// TIA Portal V17 export
// export: Created 2025-08-05T09:36:00.4025579Z, ExportSetting WithDefaults, DisplayName Totally Integrated Automation Portal, DisplayVersion V17, DisplayName TIA Portal Openness, DisplayVersion V17, DisplayName TIA Portal Version Control Interface, DisplayVersion V17, DisplayName SINAMICS Startdrive Advanced, DisplayVersion V17, DisplayName SINAMICS Startdrive G130, G150, S120, S150, SINAMICS MV, S210, DisplayVersion V17, DisplayName SINAMICS Startdrive G110M, G120, G120C, G120D, G120P, G115D, DisplayVersion V17, DisplayName STEP 7 Professional, DisplayVersion V17, DisplayName STEP 7 Safety, DisplayVersion V17, DisplayName WinCC Advanced, DisplayVersion V17
TYPE "typeHmiCounter"
TITLE = HMI part counter / HMI Stückzähler
// HMI Stückzähler [V 01.01 | Kernel_V2]
// stored: IsFailsafeCompliant false
   STRUCT
      count : Bool;   // Zählimpuls / Count pulse
      countValue : Byte;   // Anzahl der zu zählenden Gesamtteile (Gut- und Schlechtteile) / Number of parts that are counted
      countValueBad : Byte;   // Anzahl der zu zählenden Schlechtteile / Number of parts that are counted
      typIndex : Word;   // Index des Werkstücktyps, der gezählt werden soll. Bei Wert = 0 wird nur der Gesamtstückzähler berücksichtigt. Werte kleiner 0 haben eine Fehlermeldung zur Folge.
   END_STRUCT;
END_TYPE
